            !Motions to pick up bushings, if the drawers are changed, these rob targets will need changed manually
            IF currentDrawer_800=3
            THEN
                !Code below allows the X and Y axis variables to be set to allow columns to sequence
                !Movement is front to back, and left to right, starting from the front left corner
                MoveJ BP_Tray3_App10,v800,z10,gripper\WObj:=wobj_Bushing;
                IF drawer3Tray2Active
                THEN
                    MoveL Offs(BP_Tray3_App20,(currentCol)*tray3YOffset,tray3ZOffset_2,-(currentRow-1)*tray3XOffset-tray3X2Offset),v800,z10,gripper\WObj:=wobj_Bushing;
                    MoveL Offs(BP_Tray3_Pick_Back,-(currentRow-1)*tray3XOffset,(currentCol)*tray3YOffset,tray3ZOffset_2),v800,fine,gripper\WObj:=wobj_Tray3_Back;
                    Grip;
                    MoveL Offs(BP_Tray3_Dep10,(currentCol)*tray3YOffset,tray3ZOffset_2,-(currentRow-1)*tray3XOffset-tray3X2Offset),v800,fine,gripper\WObj:=wobj_Bushing;
                ELSE
                    MoveL Offs(BP_Tray3_App20,(currentCol)*tray3YOffset,tray3ZOffset_1,-(currentRow-1)*tray3XOffset),v800,z10,gripper\WObj:=wobj_Bushing;
                    MoveL Offs(BP_Tray3_Pick_Front,-(currentRow-1)*tray3XOffset,(currentCol)*tray3YOffset,tray3ZOffset_1),v800,fine,gripper\WObj:=wobj_Tray3_Front;
                    Grip;
                    MoveL Offs(BP_Tray3_Dep10,(currentCol)*tray3YOffset,tray3ZOffset_1,-(currentRow-1)*tray3XOffset),v800,fine,gripper\WObj:=wobj_Bushing;
                ENDIF
                IF Gripper_BushingPresent=1
                THEN
                    MoveL BP_Tray3_Dep20,v800,fine,gripper\WObj:=wobj_Bushing;
                ELSE
                    startIndex:=updateValidTargetPoint(tray3Index);
                    endIndex:=tray3MaxIndex;
                    endBushingFilled:=checkEndPos();
                    IF endBushingFilled=FALSE
                    THEN
                        SwitchTrayCount:=SwitchTrayCount+1;
                    ELSE
                        SwitchTrayCount:=0;
                    ENDIF
                    retryBushing:=TRUE;
                ENDIF

            ELSEIF currentDrawer_800=6
            THEN
                !Code below allows the X and Y axis variables to be set to allow columns (14 total) and rows (10 total) to sequence
                !Movement is front to back, and left to right, starting from the front left corner
                MoveJ BP_Tray6_App10,v800,z10,gripper\WObj:=wobj_Bushing;
                IF drawer6Tray2Active
                THEN
                    MoveL Offs(BP_Tray6_App20,(currentCol)*tray6YOffset,tray6ZOffset_2,-(currentRow-1)*tray6XOffset-tray6X2Offset),v800,z10,gripper\WObj:=wobj_Bushing;
                    MoveL Offs(BP_Tray6_Pick_Back,-(currentRow-1)*tray6XOffset,(currentCol)*tray6YOffset,tray6ZOffset_2),v800,fine,gripper\WObj:=wobj_Tray6_Back;
                    Grip;
                    MoveL Offs(BP_Tray6_Dep10,(currentCol)*tray6YOffset,tray6ZOffset_2,-(currentRow-1)*tray6XOffset-tray6X2Offset),v800,fine,gripper\WObj:=wobj_Bushing;
                ELSE
                    MoveL Offs(BP_Tray6_App20,(currentCol)*tray6YOffset,tray6ZOffset_1,-(currentRow-1)*tray6XOffset),v800,z10,gripper\WObj:=wobj_Bushing;
                    MoveL Offs(BP_Tray6_Pick_Front,-(currentRow-1)*tray6XOffset,(currentCol)*tray6YOffset,tray6ZOffset_1),v800,fine,gripper\WObj:=wobj_Tray6_Front;
                    Grip;
                    MoveL Offs(BP_Tray6_Dep10,(currentCol)*tray6YOffset,tray6ZOffset_1,-(currentRow-1)*tray6XOffset),v800,fine,gripper\WObj:=wobj_Bushing;
                ENDIF

                IF Gripper_BushingPresent=1
                THEN
                    MoveL BP_Tray6_Dep20,v800,fine,gripper\WObj:=wobj_Bushing;
                ELSE
                    startIndex:=updateValidTargetPoint(tray6Index);
                    endIndex:=tray6MaxIndex;
                    endBushingFilled:=checkEndPos();
                    IF endBushingFilled=FALSE
                    THEN
                        SwitchTrayCount:=SwitchTrayCount+1;
                    ELSE
                        SwitchTrayCount:=0;
                    ENDIF
                    retryBushing:=TRUE;
                ENDIF
            ENDIF

            !Incriment the current tray index to the next position
            IncrimentDrawerLocation(currentDrawer_800);

            SwitchTraysPickLocation2:
            IF endBushingFilled
            THEN
                !We can do the merge sort algorithm
                mergeSortTray;
                !Tray index has been set so go to retrypickup
                endBushingFilled:=FALSE;
                retryBushing:=TRUE;
                IF (tray3Index=-1 OR tray6Index=-1)
                THEN
                    endBushingFilled:=FALSE;
                    retryBushing:=TRUE;
                    GOTO SwitchTraysPickLocation2;
                ENDIF
                GOTO RetryPickup;
            ELSEIF retryBushing
            THEN
                !We should switch to the next tray or drawer
                IF currentDrawer_800=3 AND drawer3Tray2Active
                THEN
                    drawer3Tray2Active:=FALSE;
                    SwitchTrays(currentDrawer_800);
                ELSEIF currentDrawer_800=6 AND drawer6Tray2Active
                THEN
                    drawer6Tray2Active:=FALSE;
                    SwitchTrays(currentDrawer_800);
                ELSEIF currentDrawer_800=3
                THEN
                    drawer3Tray2Active:=TRUE;
                    Tray3Index:=0;
                ELSEIF currentDrawer_800=6
                THEN
                    drawer6Tray2Active:=TRUE;
                    Tray6Index:=0;
                ENDIF
                !If there are no bushings left at all we need to fail the part number and move on to the next part
                IF SwitchTrayCount<8
                THEN
                    IF SwitchTrayCount=4
                    THEN
                        !Call the operator
                        PulseDO\PLength:=3,Audible;
                    ENDIF
                    GOTO RetryPickup;
                ELSE
                    failedBushingFamilies{3}:=TRUE;
                    Close_All_Drawers(0);
                ENDIF
            ENDIF
        ENDIF
    ENDPROC

    !This function assumes that only one drawer is open, only use it if you are certain that the other drawers could not be open so that robot does not crash
    PROC MoveToBushingHome()
        IF Bushing_Drawer_1=1
        THEN
            MoveJ Offs(Bushing_Home,0,-TraySeparation*5,0),V1000,fine,gripper\WObj:=wobj_Bushing;
        ELSEIF Bushing_Drawer_2=1
        THEN
            MoveJ Offs(Bushing_Home,0,-TraySeparation*4,0),V1000,fine,gripper\WObj:=wobj_Bushing;
        ELSEIF Bushing_Drawer_3=1
        THEN
            MoveJ Offs(Bushing_Home,0,-TraySeparation*3,0),V1000,fine,gripper\WObj:=wobj_Bushing;
        ELSEIF Bushing_Drawer_4=1
        THEN
            MoveJ Offs(Bushing_Home,0,-TraySeparation*2,0),V1000,fine,gripper\WObj:=wobj_Bushing;
        ELSEIF Bushing_Drawer_5=1
        THEN
            MoveJ Offs(Bushing_Home,0,-TraySeparation*1,0),V1000,fine,gripper\WObj:=wobj_Bushing;
        ELSEIF Bushing_DRawer_6=1
        THEN
            MoveJ Offs(Bushing_Home,0,-TraySeparation*0,0),V1000,fine,gripper\WObj:=wobj_Bushing;
        ELSE
            !Something is wrong so stop here
            UpdateTP("ERROR: Could not move to bushing home because no tray was open");
            PrintTP;
        ENDIF
    ENDPROC

    PROC BushingPickupPointAdjustment()
        VAR num selectedTest;
        VAR btnres responseSelection;
        CONST listitem testOptions{10}:=[["","1: Test Drawer 1 Locations"],["","2: Test Drawer 2 Locations"],["","3: Test Drawer 3 Locations"],
            ["","4: Test Drawer 4 Locations"],["","5: Test Drawer 5 Locations"],["","6: Test Drawer 6 Locations"],["","7: Pick all 400 bushings"],["","8: Pick all 600 bushings"],["","9: Pick all 800 bushings"],["","10: Custom Test (Requires code input)"]];
        !Put up a message about how this is a test feature only, make sure drawers are in expected position before running test
        ErrLog 4800,"Bush-Cab Test","This is a test feature for the bushing cabinet","Please run in manual mode only","Make sure bushing drawers are in safe / expected locations","Allows for rob target changing, may require manual offset update";

        WaitTime .5;

        !Once they accept the error message we can ask them which drawer's points they would like to test
        selectedTest:=UIListView(\Result:=responseSelection\Header:="Which test would you like to run?",testOptions\Buttons:=btnOKCancel\Icon:=iconInfo\DefaultIndex:=1);

        IF responseSelection=resOK
        THEN
            IF selectedTest=1
            THEN
                !Close all drawers and open the current one
                MoveJ Offs(Bushing_Home,0,-TraySeparation*5,0),v200,fine,gripper\WObj:=wobj_Bushing;
                Close_All_Drawers(0);
                MoveJ Offs(Bushing_Home,0,-TraySeparation*5,0),v200,fine,gripper\WObj:=wobj_Bushing;
                Open_Drawer(selectedTest);
                Release;

                !The Open_Drawer function leaves the robot at Bushing_Home
                !Begin test
                MoveJ BP_Tray1_App10,v100,fine,gripper\WObj:=wobj_Bushing;
                Stop;
                MoveL BP_Tray1_App20,v50,fine,gripper\WObj:=wobj_Bushing;
                Stop;
                MoveL BP_Tray1_Pick_Front,v50,fine,gripper\WObj:=wobj_Tray1_Front;
                Stop;
                Grip;
                Stop;
                MoveL BP_Tray1_Dep10,v50,fine,gripper\WObj:=wobj_Bushing;
                Stop;
                MoveJ BP_Tray1_Dep20,v100,fine,gripper\WObj:=wobj_Bushing;
                Stop;
                MoveJ Offs(Bushing_Home,0,-TraySeparation*5,0),v200,fine,gripper\WObj:=wobj_Bushing;
                Stop;
                Release;
                !Adjust back tray
                Stop;
                MoveJ BP_Tray1_App10,v100,fine,gripper\WObj:=wobj_Bushing;
                Stop;
                MoveL BP_Tray1_App20,v50,fine,gripper\WObj:=wobj_Bushing;
                Stop;
                MoveL BP_Tray1_Pick_Back,v50,fine,gripper\WObj:=wobj_Tray1_Back;
                Stop;
                Grip;
                Stop;
                Release;
                Stop;
                MoveL BP_Tray1_App20,v50,fine,gripper\WObj:=wobj_Bushing;
                Stop;

                MoveJ BP_Tray1_App10,v100,fine,gripper\WObj:=wobj_Bushing;
                MoveL BP_Tray1_App20,v50,fine,gripper\WObj:=wobj_Bushing;
                MoveL BP_Tray1_Pick_Front,v50,fine,gripper\WObj:=wobj_Tray1_Front;
                Grip;
                MoveL BP_Tray1_Dep10,v50,fine,gripper\WObj:=wobj_Bushing;
                MoveJ BP_Tray1_Dep20,v100,fine,gripper\WObj:=wobj_Bushing;
                MoveJ Offs(Bushing_Home,0,-TraySeparation*5,0),v200,fine,gripper\WObj:=wobj_Bushing;
                Release;

                ErrLog 4800,"Test Completed","Please reset the robot and cell","Make sure to PP to main","","";
            ELSEIF selectedTest=2
            THEN
                !Close all drawers and open the current one
                MoveJ Offs(Bushing_Home,0,-TraySeparation*4,0),v200,fine,gripper\WObj:=wobj_Bushing;
                Close_All_Drawers(0);
                MoveJ Offs(Bushing_Home,0,-TraySeparation*4,0),v200,fine,gripper\WObj:=wobj_Bushing;
                Open_Drawer(selectedTest);
                Release;

                !The Open_Drawer function leaves the robot at Bushing_Home
                !Begin test
                MoveJ BP_Tray2_App10,v100,fine,gripper\WObj:=wobj_Bushing;
                Stop;
                MoveL BP_Tray2_App20,v50,fine,gripper\WObj:=wobj_Bushing;
                Stop;
                MoveL BP_Tray2_Pick_Front,v50,fine,gripper\WObj:=wobj_Tray2_Front;
                Stop;
                Grip;
                Stop;
                MoveL BP_Tray2_Dep10,v50,fine,gripper\WObj:=wobj_Bushing;
                Stop;
                MoveJ BP_Tray2_Dep20,v100,fine,gripper\WObj:=wobj_Bushing;
                Stop;
                MoveJ Offs(Bushing_Home,0,-TraySeparation*4,0),v200,fine,gripper\WObj:=wobj_Bushing;
                Stop;
                Release;
                Stop;

                MoveJ BP_Tray2_App10,v100,fine,gripper\WObj:=wobj_Bushing;
                MoveL BP_Tray2_App20,v50,fine,gripper\WObj:=wobj_Bushing;
                MoveL BP_Tray2_Pick_Front,v50,fine,gripper\WObj:=wobj_Tray2_Front;
                Grip;
                MoveL BP_Tray2_Dep10,v50,fine,gripper\WObj:=wobj_Bushing;
                MoveJ BP_Tray2_Dep20,v100,fine,gripper\WObj:=wobj_Bushing;
                MoveJ Offs(Bushing_Home,0,-TraySeparation*4,0),v200,fine,gripper\WObj:=wobj_Bushing;
                Release;

                ErrLog 4800,"Test Completed","Please reset the robot and cell","Make sure to PP to main","","";
            ELSEIF selectedTest=3
            THEN
                !Close all drawers and open the current one
                MoveJ Offs(Bushing_Home,0,-TraySeparation*3,0),v200,fine,gripper\WObj:=wobj_Bushing;
                Close_All_Drawers(0);
                MoveJ Offs(Bushing_Home,0,-TraySeparation*3,0),v200,fine,gripper\WObj:=wobj_Bushing;
                Open_Drawer(selectedTest);
                Release;

                !The Open_Drawer function leaves the robot at Bushing_Home
                !Begin test
                MoveJ BP_Tray3_App10,v100,fine,gripper\WObj:=wobj_Bushing;
                Stop;
                MoveL BP_Tray3_App20,v50,fine,gripper\WObj:=wobj_Bushing;
                Stop;
                MoveL BP_Tray3_Pick_Front,v50,fine,gripper\WObj:=wobj_Tray3_Front;
                Stop;
                Grip;
                Stop;
                MoveL BP_Tray3_Dep10,v50,fine,gripper\WObj:=wobj_Bushing;
                Stop;
                MoveJ BP_Tray3_Dep20,v100,fine,gripper\WObj:=wobj_Bushing;
                Stop;
                MoveJ Offs(Bushing_Home,0,-TraySeparation*3,0),v200,fine,gripper\WObj:=wobj_Bushing;
                Stop;
                Release;
                !Adjust back tray
                Stop;
                MoveJ BP_Tray3_App10,v100,fine,gripper\WObj:=wobj_Bushing;
                Stop;
                MoveL BP_Tray3_App20,v50,fine,gripper\WObj:=wobj_Bushing;
                Stop;
                MoveL BP_Tray3_Pick_Back,v50,fine,gripper\WObj:=wobj_Tray3_Back;
                Stop;
                Grip;
                Stop;
                Release;
                Stop;
                MoveL BP_Tray3_App20,v50,fine,gripper\WObj:=wobj_Bushing;
                Stop;

                MoveJ BP_Tray3_App10,v100,fine,gripper\WObj:=wobj_Bushing;
                MoveL BP_Tray3_App20,v50,fine,gripper\WObj:=wobj_Bushing;
                MoveL BP_Tray3_Pick_Front,v50,fine,gripper\WObj:=wobj_Tray3_Front;
                Grip;
                MoveL BP_Tray3_Dep10,v50,fine,gripper\WObj:=wobj_Bushing;
                MoveJ BP_Tray3_Dep20,v100,fine,gripper\WObj:=wobj_Bushing;
                MoveJ Offs(Bushing_Home,0,-TraySeparation*3,0),v200,fine,gripper\WObj:=wobj_Bushing;
                Release;

                ErrLog 4800,"Test Completed","Please reset the robot and cell","Make sure to PP to main","","";
            ELSEIF selectedTest=4
            THEN
                !Close all drawers and open the current one
                MoveJ Offs(Bushing_Home,0,-TraySeparation*2,0),v200,fine,gripper\WObj:=wobj_Bushing;
                Close_All_Drawers(0);
                MoveJ Offs(Bushing_Home,0,-TraySeparation*2,0),v200,fine,gripper\WObj:=wobj_Bushing;
                Open_Drawer(selectedTest);
                Release;

                !The Open_Drawer function leaves the robot at Bushing_Home
                !Begin test
                MoveJ BP_Tray4_App10,v100,fine,gripper\WObj:=wobj_Bushing;
                Stop;
                MoveL BP_Tray4_App20,v50,fine,gripper\WObj:=wobj_Bushing;
                Stop;
                MoveL BP_Tray4_Pick_Front,v50,fine,gripper\WObj:=wobj_Tray4_Front;
                Stop;
                Grip;
                Stop;
                MoveL BP_Tray4_Dep10,v50,fine,gripper\WObj:=wobj_Bushing;
                Stop;
                MoveJ BP_Tray4_Dep20,v100,fine,gripper\WObj:=wobj_Bushing;
                Stop;
                MoveJ Offs(Bushing_Home,0,-TraySeparation*2,0),v200,fine,gripper\WObj:=wobj_Bushing;
                Stop;
                Release;
                !Adjust back tray
                Stop;
                MoveJ BP_Tray4_App10,v100,fine,gripper\WObj:=wobj_Bushing;
                Stop;
                MoveL BP_Tray4_App20,v50,fine,gripper\WObj:=wobj_Bushing;
                Stop;
                MoveL BP_Tray4_Pick_Back,v50,fine,gripper\WObj:=wobj_Tray4_Back;
                Stop;
                Grip;
                Stop;
                Release;
                Stop;
                MoveL BP_Tray4_App20,v50,fine,gripper\WObj:=wobj_Bushing;
                Stop;

                MoveJ BP_Tray4_App10,v100,fine,gripper\WObj:=wobj_Bushing;
                MoveL BP_Tray4_App20,v50,fine,gripper\WObj:=wobj_Bushing;
                MoveL BP_Tray4_Pick_Front,v50,fine,gripper\WObj:=wobj_Tray4_Front;
                Grip;
                MoveL BP_Tray4_Dep10,v50,fine,gripper\WObj:=wobj_Bushing;
                MoveJ BP_Tray4_Dep20,v100,fine,gripper\WObj:=wobj_Bushing;
                MoveJ Offs(Bushing_Home,0,-TraySeparation*2,0),v200,fine,gripper\WObj:=wobj_Bushing;
                Release;

                ErrLog 4800,"Test Completed","Please reset the robot and cell","Make sure to PP to main","","";
            ELSEIF selectedTest=5
            THEN
                !Close all drawers and open the current one
                MoveJ Offs(Bushing_Home,0,-TraySeparation*1,0),v200,fine,gripper\WObj:=wobj_Bushing;
                Close_All_Drawers(0);
                MoveJ Offs(Bushing_Home,0,-TraySeparation*1,0),v200,fine,gripper\WObj:=wobj_Bushing;
                Open_Drawer(selectedTest);
                Release;

                !The Open_Drawer function leaves the robot at Bushing_Home
                !Begin test
                MoveJ BP_Tray5_App10,v100,fine,gripper\WObj:=wobj_Bushing;
                Stop;
                MoveL BP_Tray5_App20,v50,fine,gripper\WObj:=wobj_Bushing;
                Stop;
                MoveL BP_Tray5_Pick_Front,v50,fine,gripper\WObj:=wobj_Tray5_Front;
                Stop;
                Grip;
                Stop;
                MoveL BP_Tray5_Dep10,v50,fine,gripper\WObj:=wobj_Bushing;
                Stop;
                MoveJ BP_Tray5_Dep20,v100,fine,gripper\WObj:=wobj_Bushing;
                Stop;
                MoveJ Offs(Bushing_Home,0,-TraySeparation*1,0),v200,fine,gripper\WObj:=wobj_Bushing;
                Stop;
                Release;
                Stop;

                MoveJ BP_Tray5_App10,v100,fine,gripper\WObj:=wobj_Bushing;
                MoveL BP_Tray5_App20,v50,fine,gripper\WObj:=wobj_Bushing;
                MoveL BP_Tray5_Pick_Front,v50,fine,gripper\WObj:=wobj_Tray5_Front;
                Grip;
                MoveL BP_Tray5_Dep10,v50,fine,gripper\WObj:=wobj_Bushing;
                MoveJ BP_Tray5_Dep20,v100,fine,gripper\WObj:=wobj_Bushing;
                MoveJ Offs(Bushing_Home,0,-TraySeparation*1,0),v200,fine,gripper\WObj:=wobj_Bushing;
                Release;

                ErrLog 4800,"Test Completed","Please reset the robot and cell","Make sure to PP to main","","";
            ELSEIF selectedTest=6
            THEN
                !Close all drawers and open the current one
                MoveJ Bushing_Home,v200,fine,gripper\WObj:=wobj_Bushing;
                Close_All_Drawers(0);
                MoveJ Bushing_Home,v200,fine,gripper\WObj:=wobj_Bushing;
                Open_Drawer(selectedTest);
                Release;

                !The Open_Drawer function leaves the robot at Bushing_Home
                !Begin test
                MoveJ BP_Tray6_App10,v100,fine,gripper\WObj:=wobj_Bushing;
                Stop;
                MoveL BP_Tray6_App20,v50,fine,gripper\WObj:=wobj_Bushing;
                Stop;
                MoveL BP_Tray6_Pick_Front,v50,fine,gripper\WObj:=wobj_Tray6_Front;
                Stop;
                Grip;
                Stop;
                MoveL BP_Tray6_Dep10,v50,fine,gripper\WObj:=wobj_Bushing;
                Stop;
                MoveJ BP_Tray6_Dep20,v100,fine,gripper\WObj:=wobj_Bushing;
                Stop;
                MoveJ Bushing_Home,v200,fine,gripper\WObj:=wobj_Bushing;
                Stop;
                Release;
                !Adjust back tray
                Stop;
                MoveJ BP_Tray6_App10,v100,fine,gripper\WObj:=wobj_Bushing;
                Stop;
                MoveL BP_Tray6_App20,v50,fine,gripper\WObj:=wobj_Bushing;
                Stop;
                MoveL BP_Tray6_Pick_Back,v50,fine,gripper\WObj:=wobj_Tray6_Back;
                Stop;
                Grip;
                Stop;
                Release;
                Stop;
                MoveL BP_Tray6_App20,v50,fine,gripper\WObj:=wobj_Bushing;
                Stop;

                MoveJ BP_Tray6_App10,v100,fine,gripper\WObj:=wobj_Bushing;
                MoveL BP_Tray6_App20,v50,fine,gripper\WObj:=wobj_Bushing;
                MoveL BP_Tray6_Pick_Front,v50,fine,gripper\WObj:=wobj_Tray6_Front;
                Grip;
                MoveL BP_Tray6_Dep10,v50,fine,gripper\WObj:=wobj_Bushing;
                MoveJ BP_Tray6_Dep20,v100,fine,gripper\WObj:=wobj_Bushing;
                MoveJ Bushing_Home,v200,fine,gripper\WObj:=wobj_Bushing;
                Release;

                ErrLog 4800,"Test Completed","Please reset the robot and cell","Make sure to PP to main","","";
            ELSEIF selectedTest=7 OR selectedTest=8 OR selectedTest=9
            THEN
                IF selectedTest=7
                THEN
                    partNumber:=11;
                ELSEIF selectedTest=8
                THEN
                    partNumber:=13;
                ELSEIF selectedTest=9
                THEN
                    partNumber:=15;
                ENDIF

                tray1Index:=0;
                tray2Index:=0;
                tray3Index:=0;
                tray4Index:=0;
                tray5Index:=0;
                tray6Index:=0;
                drawer1Tray2Active:=FALSE;
                drawer2Tray2Active:=FALSE;
                drawer3Tray2Active:=FALSE;
                drawer4Tray2Active:=FALSE;
                drawer5Tray2Active:=FALSE;
                drawer6Tray2Active:=FALSE;

                currentDrawer_400:=1;
                currentDrawer_600:=5;
                currentDrawer_800:=6;

                !For Loop that iterates for both drawers of parts which is 140*4=560 (Plus a few extra)
                FOR i FROM 1 TO 570 DO
                    Bushing_Pickup;
                    !Move to current home location to drop bushing
                    MoveToBushingHome;
                    Release;

                    !Incriment the bushing part counter
                    IF partNumber=11
                    THEN
                        IncrimentDrawerLocation(currentDrawer_400);
                    ELSEIF partNumber=13
                    THEN
                        IncrimentDrawerLocation(currentDrawer_600);
                    ELSEIF partNumber=15
                    THEN
                        IncrimentDrawerLocation(currentDrawer_800);
                    ENDIF
                ENDFOR
            ELSEIF selectedTest=10
            THEN
                !Put your own custom code here to test something not covered above

            ENDIF
        ENDIF
    ENDPROC
ENDMODULE
